FUNCTION_BLOCK Test_RTrimEx_HandlesTrimmingManyChars EXTENDS T_UnitTestBase
VAR_INPUT
END_VAR
VAR_OUTPUT
END_VAR
VAR
	SubjectString : T_MaxString := 'Badger';
END_VAR

Assertion.AssertEquals_STRING(
	Expected := '',
	Actual := F_RTrimEx(n := 20, str := SubjectString),
	VariableName := 'F_LTrimEx(SubjectString)');
	
TestFinished();

END_FUNCTION_BLOCK

(* stored: Version 1.1.0.1, ProductVersion 3.1.4024.6
   POU Test_RTrimEx_HandlesTrimmingManyChars: Id {7d1ecfd7-56bb-0e5e-2d68-ef19da97a9f8}, SpecialFunc None *)
